FUNCTION_BLOCK BfbIDMTCurve
  (* Standard: 61499-2 *)
  (* Version 0.1, 2019-00-29, hpea485, UOA *)
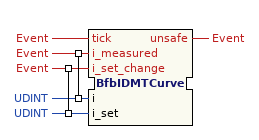
  EVENT_INPUT
    tick;
    i_measured WITH i;
    i_set_change WITH i_set;
  END_EVENT
  EVENT_OUTPUT
    unsafe;
  END_EVENT
  VAR_INPUT
    i : UDINT;
    i_set : UDINT;
  END_VAR
  VAR
    cnt : ULINT := 0;
    max : UDINT := 0.0;
    k : UDINT := 100.0;
    b : UDINT := 135;
    a : UDINT := 1.0;
  END_VAR
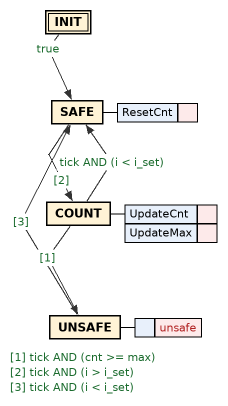
  EC_STATES
    INIT;
    SAFE : ResetCnt;
    COUNT : UpdateCnt, UpdateMax;
    UNSAFE : -> unsafe;
  END_STATES
  EC_TRANSITIONS
    INIT TO SAFE := true;
    SAFE TO COUNT := tick AND (i > i_set);
    COUNT TO UNSAFE := tick AND (cnt >= max);
    COUNT TO SAFE := tick AND (i < i_set);
    UNSAFE TO SAFE := tick AND (i < i_set);
  END_TRANSITIONS
  ALGORITHM ResetCnt IN C:
me->cnt = 0;
  END_ALGORITHM
  ALGORITHM UpdateCnt IN C:
me->cnt = me->cnt + 1;
  END_ALGORITHM
  ALGORITHM UpdateMax IN C:
me->max = (me->k * me->b) / ((me->i / me->i_set) - 1);
  END_ALGORITHM
END_FUNCTION_BLOCK
